// Mitsubishi GX Works2 project: KemNghiaDrillV1   PLC: FX3U/FX3UC

// global labels: Global1
VAR_GLOBAL
  Run AT M0 : BOOL;
  RunStop AT M1 : BOOL;
  AxisRun AT M11 : BOOL;
  AxisDirection AT M12 : BOOL;
  Drill AT M40 : BOOL;
  FoilOut AT M60 : BOOL;
  DrillN AT M41 : BOOL;
  DrillP AT M42 : BOOL;
  FoilOutN AT M61 : BOOL;
  FoilOutP AT M62 : BOOL;
  AxisTarget AT D10 : DINT;
  AxisRPM AT D14 : DINT;
  AxisCurrent AT D8360 : DINT;
  RunState AT D0 : INT;
  RunI AT X000 : BOOL;
  RunStopI AT X001 : BOOL;
  DrillNI AT X007 : BOOL;
  DrillPI AT X010 : BOOL;
  FoilOutNI AT X013 : BOOL;
  FoilOutPI AT X014 : BOOL;
  AxisPulseO AT Y002 : BOOL;
  AxisDirectionO AT Y004 : BOOL;
  FoilExtractTopO AT Y010 : BOOL;
  FoilExtractBotO AT Y011 : BOOL;
  DrillO AT Y012 : BOOL;
  FoilOutO AT Y014 : BOOL;
  AxisMinI AT X002 : BOOL;
  AxisOnO AT Y006 : BOOL;
  RunStateFoilExtract AT D1 : INT;
  RunStateFoilOut AT D4 : INT;
  RunStateDrill AT D2 : INT;
  FoilExtractTop AT M20 : BOOL;
  FoilExtractTopN AT M21 : BOOL;
  FoilExtractTopP AT M22 : BOOL;
  FoilExtractBot AT M30 : BOOL;
  FoilExtractBotN AT M31 : BOOL;
  FoilExtractBotP AT M32 : BOOL;
  FoilExtractTopPI AT X004 : BOOL;
  FoilExtractBotPI AT X006 : BOOL;
  FoilExtractTopNI AT X003 : BOOL;
  FoilExtractBotNI AT X005 : BOOL;
  EnableTapI AT X015 : BOOL;
  AxisPPR AT D12 : DINT;
  AirAO AT Y015 : BOOL;
  AirA AT M70 : BOOL;
  AxisOn AT M10 : BOOL;
  AxisBusy AT M8360 : BOOL;
  AxisAccel AT D8368 : INT;
  AxisDecel AT D8369 : INT;
  AxisInterruptReverse AT M8367 : BOOL;
  AxisTarRSkip AT D16 : INT;
  AxisTarR AT M13 : BOOL;
  IgnoreDrillTapO AT Y017 : BOOL;
END_VAR

// task Task_01 (event TRUE, interval 0, priority 31): POU_01

PROGRAM POU_01
VAR
  fFall : BOOL;
  fRise : BOOL;
  fAxisPulseFrequency : DINT;
  fTmp : BOOL;
  fRunStateNext : BOOL;
  fRunStateFoilExtractNext : BOOL;
  fRunStateDrillNext : BOOL;
  fRunStateTapNext : BOOL;
  fRunStateFoilOutNext : BOOL;
  fAxisHzPerRPM : DINT;
  fTurnStepCount : INT;
  fAxisTest : BOOL;
  fAxisDRVIOffset : DINT;
  fPs : ARRAY [0..7] OF DINT;
  fPsSet : BOOL;
  fStepReady : BOOL;
END_VAR
VAR CONSTANT
  fSectorCount : INT := 1;
END_VAR
VAR
  fAxisDRVIFrequency : DINT;
  fAxisDRVIOffsetBefore : DINT;
  fRunAuto : BOOL;
  fIgnoreDrillTap : BOOL;
END_VAR
MOV(M8002, 500, AxisAccel);
MOV(M8002, 500, AxisDecel);
SET(M8002, M8336);
MOV(M8002, HF2FF, D8336);
RST(M8002, AxisInterruptReverse);
ZRST(M8002, RunState, RunStateFoilOut);
SET(M8002, FoilExtractTop);
SET(M8002, FoilExtractBot);
RST(M8002, Drill);
RST(M8002, fAxisTest);
RST(M8002, fIgnoreDrillTap);
RST(M8002, fRunAuto);
SET(M8002, fPsSet);
DMOV(fPsSet, 6930, fPs[0]); (*use this value as pulse per sector*)
DMOV(fPsSet, 6930, fPs[1]);
DMOV(fPsSet, 13860, fPs[2]);
DMOV(fPsSet, 20790, fPs[3]);
DMOV(fPsSet, 27720, fPs[4]);
DMOV(fPsSet, 34650, fPs[5]);
DMOV(fPsSet, 41580, fPs[6]);
DMOV(fPsSet, 48510, fPs[7]);
RST(fPsSet, fPsSet);

DMOV(M8002, 150, fAxisDRVIOffset);
DMOV(M8002, 300, fAxisDRVIOffsetBefore); (*offset beforce must larger than offset*)
DMOV(M8002, 300, fAxisDRVIFrequency);

OUT_T(M8000, TC0, 50);
SET(TC0 AND Run AND RunState = 0, fTmp);
RST(fTmp, Run);
DMOV(fTmp, 55440, AxisPPR);
DMOV(fTmp, AxisPPR / 60, fAxisHzPerRPM);
DMOV(fTmp, 30, AxisRPM);
DMOV(fTmp, AxisRPM * fAxisHzPerRPM, fAxisPulseFrequency);
RST(fTmp, AxisCurrent);
MOV(fTmp, 1, RunState);
RST(fTmp, fTmp);
SET(RunStop, fTmp);
RST(fTmp, RunStop);
ZRST(fTmp, RunState, RunStateFoilOut);
ZRST(fTmp, fRunStateFoilOutNext, fRunStateNext);
RST(fTmp, AxisRun);
RST(fTmp, AxisOn);
RST(fTmp, FoilOut);
RST(fTmp, fRunAuto);
RST(fTmp, fTmp);

INC(fRunStateNext, RunState);
INC(fRunStateFoilExtractNext, RunStateFoilExtract);
INC(fRunStateDrillNext, RunStateDrill);
INC(fRunStateFoilOutNext, RunStateFoilOut);
ZRST(M8000, fRunStateFoilOutNext, fRunStateNext);
DECO(M8000, RunState, 6, M100); DECO(M8000, RunState, 6, M1000); ZRST(NOT AxisTarR, M1000, M1063);
DECO(M8000, RunStateFoilExtract, 6, M200);
DECO(M8000, RunStateDrill, 6, M300);
DECO(M8000, RunStateFoilOut, 6, M400);

(*||||||||||*)
(*turn axis on*)
OUT_T(M101, TC1, 20);
SET(M101 AND NOT AxisOn, AxisOn);
SET(M101 AND TC1, fRunStateNext);
(*move fast before ddvi*)
DMOVP(M1002, AxisCurrent + fPs[0] - fAxisDRVIOffsetBefore, AxisTarget);
SET(M1002, AxisRun);
SET(M1002, fRunStateNext);
(*setup ddvi*)
SET(M1003, fRunStateNext);
(*ddvi*)
DDVIT(M104, fAxisDRVIOffset, fAxisDRVIFrequency, AxisPulseO, AxisDirection);
SET(M104 AND M8029, fRunStateNext);
RST(M104 AND M8029, M104);
(*get origin done*)
RST(M1005, AxisCurrent);
MOV(M1005, 7, RunState);
(*start run*)
RST(M1007, fTurnStepCount);
RST(M1007, AxisCurrent);
MOV(M1007, 14, RunState);
(*move next position*)
DMOV(M1008, fPs[fTurnStepCount], AxisTarget);
SET(M1008, AxisRun);
MOV(M1008, 14, RunState);
(*move next position done*)
(*final*) SET(M1014 AND fTurnStepCount = (fSectorCount - 1), fTmp);
(*final*) INC(fTmp, fTurnStepCount);
(*final*) MOV(fTmp, 15, RunState);
(*final*) RST(fTmp, M1014);
(*final*) RST(fTmp, fTmp);
INC(M1014 AND fTurnStepCount < fSectorCount, fTurnStepCount);
(*full turn*) SET(M1014 AND fTurnStepCount >= fSectorCount, fTmp);
(*full turn*) RST(fTmp, fTurnStepCount);
(*full turn*) MOV(fTmp, 2, RunState);
(*full turn*) RST(fTmp, M1014);
(*full turn*) RST(fTmp, fTmp);
MOV(M1014, 15, RunState);
(*process, delay 500ms with TC2 before, why?*)
SET(M1015, AirA);
MOV(M1015, 1, RunStateFoilExtract);
MOV(M1015, 1, RunStateDrill);
MOV(M1015, 1, RunStateFoilOut);
SET(M1015, fRunStateNext);
(*wait all done*)
(*test*) OUT_T(M1016, TC3, 5);
(*test*) SET(M1016 AND TC3 AND fAxisTest AND fStepReady, fTmp);
(*test*) RST(fStepReady, fStepReady);
SET(M1016 AND M210 AND M310 AND M410, fTmp);
ZRST(fTmp, RunStateFoilExtract, RunStateFoilOut);
SET(fTmp, fRunStateNext);
RST(fTmp, fTmp);
(*manual step*)
SET(M1017 AND NOT fRunAuto AND Run, fRunStateNext);
SET(M1017 AND fRunAuto, fRunStateNext);
RST(Run, Run);
(**)
SET(M1018 AND fSectorCount = 1, fTmp);
MOV(fTmp, 2, RunState);
RST(fTmp, M1018);
RST(fTmp, fTmp);
SET(M1018 AND fTurnStepCount = fSectorCount, fTmp);
MOV(M1018 AND NOT fTmp, 8, RunState);
MOV(M1018 AND fTmp, 14, RunState);
RST(fTmp, fTmp);
(**)
(*||||||||||*)
(*||||||||||FoilExtract*)
(*not ready, top and bot forward*)
SET(M201 AND NOT FoilExtractTopP, FoilExtractTop);
SET(M201 AND NOT FoilExtractBotP, FoilExtractBot);
RST(M201 AND NOT (FoilExtractTopP OR FoilExtractBotP), M201);
(*ready, bot back*)
RST(M201, FoilExtractBot);
SET(M201, fRunStateFoilExtractNext);
(*bot back done, bot forward*)
RST(M202 AND NOT FoilExtractBotN, M202);
SET(M202, FoilExtractBot);
SET(M202, fRunStateFoilExtractNext);
(*bot forward done, top back*)
OUT_T(M203, TC50, 5);
SET(M203 AND TC50 AND FoilExtractBotP, fTmp);
RST(fTmp, FoilExtractTop);
SET(fTmp, fRunStateFoilExtractNext);
RST(fTmp, fTmp);
(*top back done, top forward*)
RST(M204 AND NOT FoilExtractTopN, M204);
SET(M204, FoilExtractTop);
SET(M204, fRunStateFoilExtractNext);
(*top forward done, end*)
MOV(M205 AND FoilExtractTopP, 10, RunStateFoilExtract);
(*||||||||||*)
(*||||||||||Drill*)
(**)
MOV(M301 AND fIgnoreDrillTap, 10, RunStateDrill);
SET(M301 AND NOT fIgnoreDrillTap, fRunStateDrillNext);
(**)
SET(M302 AND DrillN, fRunStateDrillNext);
(**)
SET(M303, Drill);
SET(M303, fRunStateDrillNext);
(**)
SET(M304 AND NOT DrillN AND DrillP, fRunStateDrillNext);
(**)
MOV(M305 AND NOT DrillP AND DrillN, 10, RunStateDrill);
(*||||||||||*)
(*||||||||||FoilOut*)
(**)
RST(M401 AND NOT FoilOutN, FoilOut);
SET(M401 AND FoilOutN, fRunStateFoilOutNext);
(**)
SET(M402, FoilOut);
SET(M402, fRunStateFoilOutNext);
(**)
RST(M403 AND FoilOutP, FoilOut);
SET(M403 AND FoilOutP, fRunStateFoilOutNext);
(*down done, end*)
MOV(M404 AND FoilOutN, 10, RunStateFoilOut);
(*||||||||||*)

(*||||||||||*)
RST(AxisRun AND AxisTarget = AxisCurrent, AxisRun);
DDRVA(AxisRun, AxisTarget, fAxisPulseFrequency, AxisPulseO, AxisDirection);
RST(M8029, AxisRun);
OUT(AxisDirection, AxisDirectionO);
INC(NOT AxisRun AND NOT AxisBusy AND AxisTarRSkip < 5, AxisTarRSkip);
RST(AxisRun, AxisTarRSkip);
OUT(AxisTarRSkip >= 5, AxisTarR);
(*||||||||||*)

(*Input*)
PLS(RunI, fRise); SET(fRise, Run);
PLS(RunStopI, fRise); SET(fRise, RunStop);
OUT_T(RunI, TC4, 20); SET(TC4, fRunAuto);
OUT_T(RunStopI AND NOT fIgnoreDrillTap, TC5, 20); SET(TC5, fIgnoreDrillTap);
OUT_T(RunStopI AND fIgnoreDrillTap, TC6, 20); RST(TC6, fIgnoreDrillTap);

(**)
OUT_T(NOT FoilExtractTop, TC10, 10); SET(TC10, FoilExtractTopN); RST(TC10, FoilExtractTopP);
OUT_T(FoilExtractTop, TC11, 3); SET(TC11, FoilExtractTopP); RST(TC11, FoilExtractTopN);
(**)
OUT_T(NOT FoilExtractBot, TC12, 10); SET(TC12, FoilExtractBotN); RST(TC12, FoilExtractBotP);
OUT_T(FoilExtractBot, TC13, 3); SET(TC13, FoilExtractBotP); RST(TC13, FoilExtractBotN);
(**)

(**)
PLS(DrillNI, fRise); SET(fRise, DrillN); RST(fRise, DrillP);
PLS(DrillPI, fRise); SET(fRise, DrillP); RST(fRise, DrillN);
SET(DrillNI, DrillN); RST(DrillNI, DrillP);
SET(DrillPI, DrillP); RST(DrillPI, DrillN);
(**)

(**)
OUT_T(FoilOutNI, TC18, 3); SET(TC18, FoilOutN); RST(TC18, FoilOutP);
OUT_T(FoilOutPI, TC19, 3); SET(TC19, FoilOutP); RST(TC19, FoilOutN);
(**)

(*Output*)
OUT_T(AirA, TC20, 10); RST(TC20, AirA);
OUT_T(Drill, TC21, 2); RST(TC21, Drill);
(**)
OUT(AxisOn, AxisOnO);
OUT(NOT FoilExtractTop, FoilExtractTopO);
OUT(NOT FoilExtractBot, FoilExtractBotO);
OUT(Drill, DrillO);
OUT(FoilOut, FoilOutO);
OUT(AirA, AirAO);
OUT(fIgnoreDrillTap, IgnoreDrillTapO);
END_PROGRAM
